(* Logix 5000 project; controller ktc_exapmple2 vendor 1 type 14 code 150 rev 30.11; software revision 30.00 *)

TASK MainTask (continuous, watchdog 500 ms) : MainProgram

MODULES
   Local : vendor 1 type 14 code 150 (Compact 0, rev 30.11)
      Counters : Embedded (Compact 3, rev 1.1, Output RPI 20 ms)
      Discrete_IO : Embedded (Compact 1, rev 3.1, Output RPI 20 ms)
      Analog_IO : Embedded (Compact 2, rev 1.1, Output RPI 80 ms)
END_MODULES

PROGRAM MainProgram   (* main routine MainRoutine *)
VAR
   LED_1 : BOOL;
   PB_3 : ALIAS FOR Local:1:I.Data.0;   // PUSH BUTTON NO 6
   PL_1 : ALIAS FOR Local:1:O.Data.7;   // LED 7
   PL_2 : ALIAS FOR Local:1:O.Data.1;   // LED1
   PL_3 : ALIAS FOR Local:1:O.Data.3;   // LED 3
   PL_4 : ALIAS FOR Local:1:O.Data.6;   // LED 6
   SW_1 : ALIAS FOR Local:1:I.Data.4;   // SWITCH
END_VAR

ROUTINE MainRoutine   (* ladder *)
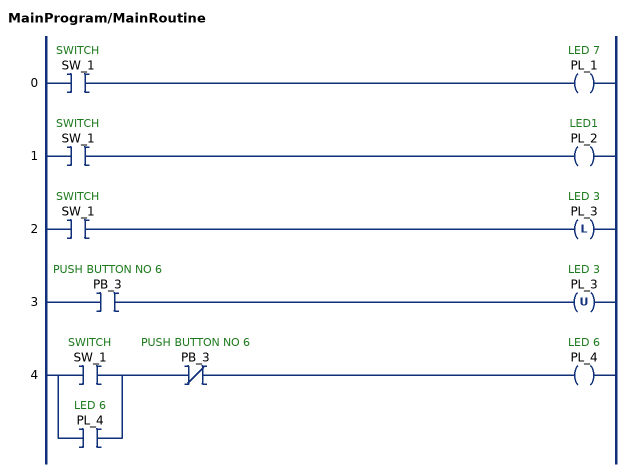
   0: XIC(SW_1)OTE(PL_1);
   1: XIC(SW_1)OTE(PL_2);
   2: XIC(SW_1)OTL(PL_3);
   3: XIC(PB_3)OTU(PL_3);
   4: [XIC(SW_1) ,XIC(PL_4) ]XIO(PB_3)OTE(PL_4);
END_ROUTINE
END_PROGRAM
